Fanuc KAREL source: kb00064.KL

-- PROVISIONAL review KL for V1013-1; original PC SHA256 a6142224ad8e64f01068c77203347739412ebf1c77324823da05ca82c5abd815
-- Incomplete behavior may be omitted. Consult companion uncertainty JSON. Do not deploy.
PROGRAM KB00064
%NOLOCKGROUP
BEGIN
  -- UNRESOLVED_PC offsets 5-14; opcodes 3F,75
  -- UNRESOLVED_PC offsets 19-28; opcodes 3F,75
  -- UNRESOLVED_PC offsets 33-40; opcodes 9D,23
  -- UNRESOLVED_PC offsets 45-71; opcodes 27,22,2A,22,2A,22,31
  -- UNRESOLVED_PC offsets 76-80; opcodes 7F
END KB00064
